// Mitsubishi GX Works2 project: ch4   PLC: FX3U/FX3UC

PROGRAM MAIN
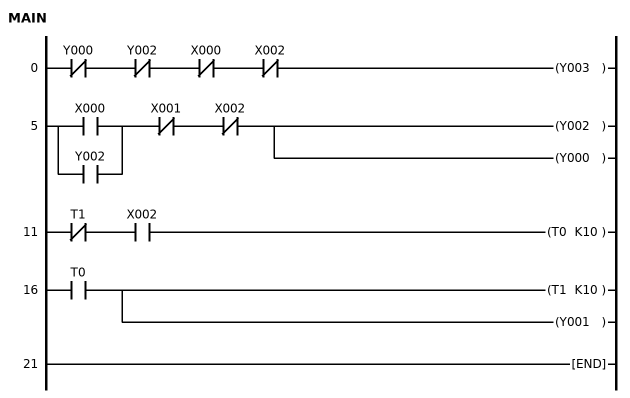
0     LDI     Y000
      ANI     Y002
      ANI     X000
      ANI     X002
      OUT     Y003
5     LD      X000
      OR      Y002
      ANI     X001
      ANI     X002
      OUT     Y002
      OUT     Y000
11    LDI     T1
      AND     X002
      OUT     T0 K10
16    LD      T0
      OUT     T1 K10
      OUT     Y001
21    END
END_PROGRAM
